// TIA Portal V17 export
// export: Created 2024-09-02T12:50:30.8652748Z, ExportSetting WithDefaults, DisplayName Totally Integrated Automation Portal, DisplayVersion V17, DisplayName TIA Portal Openness, DisplayVersion V17, DisplayName TIA Portal Version Control Interface, DisplayVersion V17, DisplayName STEP 7 Professional, DisplayVersion V17, DisplayName STEP 7 Safety, DisplayVersion V17, DisplayName WinCC Professional, DisplayVersion V17
TYPE "TypeEthernetVerbStatus"
// stored: IsFailsafeCompliant false
   STRUCT
      InterfaceId : UInt;
      ID : Word;
      ConnectionType : Byte;
      ActiveEstablished : Bool;
      State : Byte;
      Kind : Byte;
      SentBytes : UDInt;
      ReceivedBytes : UDInt;
      ConnTrials : UDInt;
      ConnTrialsSuccess : UDInt;
      LastConnErrReason : UDInt;
      LastConnErrTimeStamp : LDT;
      LastDisconnReason : UDInt;
      LastDisconnTimeStamp : LDT;
   END_STRUCT;
END_TYPE
